Staubli VAL3: updateCycleNum.pgx

program updateCycleNum(num x_nNum (dimensions=1))
  local num l_nLocalWord[2]
begin

  //let's suppose that in the plc's db "nDBwrite" there is a word, starting from byte 10, that represent the number of cyle performed by
  //the robot

  //first of all we have to "translate" the argument x_nNum in a 2 byte buffer representing the word (using "big-endian" format)
  //the better way to do this is a local 2 elements array written by the "helper" function setWordAt
  call S7:setWordAt(0,x_nNum,l_nLocalWord)

  //then we write this buffer to nDBwrite!
  call S7:writeArea(S7:nAreaDB,nDBwrite,l_nLocalWord,0,size(l_nLocalWord))

end
